# B&R Automation Studio project Cognex_V1_5
Automation Studio 4.0.21.35 SP

## Configuration PP500_15

CPU , AutomationRuntime H4.06, Build 4.1.2, Vc V4.05.6, Safety 1.6

### Hardware
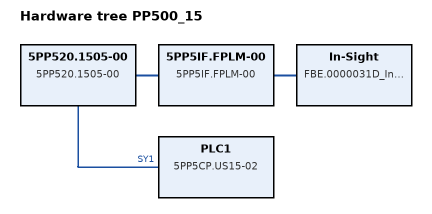
```
5PP520.1505-00 : 5PP520.1505-00 v2.0.1.1
  Connector IF3:
    ActivateDevice = 1
    Mode = DHCP Server
    InternetAddress = 192.168.0.10
    SubnetMask = 255.255.255.0
    Lease1
    LeaseName1 = loc
    LeaseStartAddress1 = 192.168.0.220
    LeaseStopAddress1 = 192.168.0.230
    LeaseSubnetMask1 = 255.255.255.0
    Vnc1
    VncVcObjectName1 = Visu
    VncPortNumber1 = 5900
    VncMaxConnections1 = 1
    VncRefreshRate1 = 1000
    VncConnectionTimeout1 = 4
    VncAuthentication1 = 1
    VncPasswordViewOnly1 = r
    VncPasswordViewControl1 = w
  VcObjectName = Visu
5PP5IF.FPLM-00 : 5PP5IF.FPLM-00 v2.1.3.0  [SL -> 5PP520.1505-00.SL1]
  Connector IF1:
    MtuSize = 1500
    CycleTime = 400
    InternetAddress = 10.49.40.10
    SubnetMask = 255.255.255.0
In-Sight : FBE.0000031D_In-Sight-7000 v1.0 (OrderNumber=In-Sight)  [PLK1 -> 5PP5IF.FPLM-00.IF1 (NodeNumber=1)]
  Supervision = off
  p2000s01_direction = wo
  p2000s02_direction = wo
  p2001s01_direction = ro
  p2001s02_direction = ro
  p2010s01_direction = ro
  p2011s01_direction = ro
  p2011s02_direction = ro
  p2011s03_direction = ro
  p2011s04_direction = ro
  p2011s05_direction = ro
  p2011s06_direction = ro
  p2011s07_direction = ro
  p2011s08_direction = ro
  p2011s09_direction = ro
  p2011s0A_direction = ro
  p2011s0B_direction = ro
  p2021s01_direction = wo
  p2021s02_direction = wo
  p2021s03_direction = wo
PLC1 : 5PP5CP.US15-02 v2.0.3.0  [SY -> 5PP520.1505-00.SY1]
  PreserveNonVolatileSystemSettings = 0
  Connections = 8
  TimerDeviceType = EPLX2X
  TaskClassIdleTime = 800
  Cyclic1Duration = 2000
  Cyclic1Tolerance = 2000
  Cyclic1Stack = 65535
  Cyclic2Stack = 65535
  Cyclic3Stack = 65535
  Cyclic4Stack = 65535
  Cyclic5Stack = 65535
  Cyclic6Stack = 65535
  Cyclic7Stack = 65535
  Cyclic8Duration = 4000
  Cyclic8Stack = 65535
  TimerDevice = 5PP5IF.FPLM-00.IF1
```

## Configuration X20CPU1484

CPU , AutomationRuntime V3.08, Build 4.1.2, Vc V3.95.6

## Logical view

Binary libraries used (declarations not repeated): Operator, Runtime, AsTime, AsIecCon, sys_lib, asstring, FileIO, Visapi, AsTCP, AsICMP, standard, BR_ATL_LOG, BR_ATL_BMP, BR_ATL_COG


- Program Logical/Cognex (IEC) - Cognex IO mapping (no source held here)

### Program Logical/CognexVisCommissioning (IEC) - Cognex camera commissioning

#### CognexVisCommissioning.var
```iecst
(*-------------------------------------------------------------------------------------------------------------------------------------------------------------------------------------------------------------------------*)
VAR
	data : ARRAY[0..999] OF USINT; (*Send and receive buffer (size must be even)*)
	data_string : ARRAY[0..19] OF STRING[80]; (*Receive data split up as string*)
	NativeModeCommandStatus : INT;
	NaticeModeCommand : USINT;
	NativeModeCommand_0 : NativeModeCommand;
	NativeModeWriteFile_0 : NativeModeWriteFile;
	DirCreate_0 : DirCreate;
	DevLink_0 : DevLink;
	TransferProgressStatus : UINT;
	vsTransferProgress : USINT;
END_VAR
(*--------------------------------------------------------------------------------------------------------------------------------------------------------------------------------------------------------------------------------------------*)
VAR
	vkNativeModeConnect : BOOL;
	NativeModeLoggedIn : UINT;
	NativeModeStatus : UINT;
	NativeModeLogin_0 : NativeModeLogin;
	NativeModeLogout_0 : NativeModeLogout;
END_VAR
(*--------------------------------------------------------------------------------------------------------------------------------------------------------------------------------------------------------------------------------------------*)
VAR
	vkTransferWrite : USINT;
	vsErrorReset : UINT := 1;
	vkErrorReset : BOOL;
END_VAR
```

#### CognexVisCommissioning.ab
```automation-basic
(********************************************************************
 * COPYRIGHT --
 ********************************************************************
 * Author: strickers
 * Version: 1.0
 * This task has the following purpose
 * - Connect to Cognex telnet (Native interface)
 * - Read command_status information
 * - Read and write camera jobs
 * - Read and write camera settings
 ********************************************************************)

PROGRAM _INIT
	(* --------------------------------------------------------------------------------------------------------- *)
	(* Create file device for Cognex files and configuration files *)
	LOOP
		DevLink_0.enable 	= 1
		DevLink_0.pDevice 	= ADR("root")
		DevLink_0.pParam 	= ADR("/DEVICE=C:\\")
		DevLink_0 FUB DevLink()
		EXITIF(DevLink_0.status <> 65535)
	ENDLOOP
	(* --------------------------------------------------------------------------------------------------------- *)
	(* Create folder for Cognex files and configuration files *)
	LOOP
		DirCreate_0.enable 	= 1
		DirCreate_0.pDevice = ADR("root")
		DirCreate_0.pName 	= ADR("cognex_files")
		DirCreate_0 FUB DirCreate()
		EXITIF(DirCreate_0.status <> 65535)
	ENDLOOP
	(* --------------------------------------------------------------------------------------------------------- *)
	(* Create file device for Cognex files and configuration files *)
	LOOP
		DevLink_0.enable 	= 1
		DevLink_0.pDevice 	= ADR("CognexFiles")
		DevLink_0.pParam 	= ADR("/DEVICE=C:\\cognex_files")
		DevLink_0 FUB DevLink()
		EXITIF(DevLink_0.status <> 65535)
	ENDLOOP
	NativeModeStatus = VIS_INACTIVE
	TransferProgressStatus = VIS_HIDDEN
END_PROGRAM

PROGRAM _CYCLIC

(* --------------------------------------------------------------------------------------------------------- *)
(* Connect to camera
(* --------------------------------------------------------------------------------------------------------- *)
IF(EDGEPOS(vkNativeModeConnect)) THEN
	NewLogEntry("Connecting to camera...", ADR(logbook), 20)
ENDIF
IF(vkNativeModeConnect = TRUE) THEN
	IF(NativeModeLoggedIn = FALSE) THEN
		NativeModeLogin_0.enable = 1
		NativeModeLogin_0.ip = ADR(CognexEthIP)
		NativeModeLogin_0 FUB NativeModeLogin()
		IF(NativeModeLogin_0.status <> 65535) THEN
			IF(NativeModeLogin_0.status = 0) THEN
				NewLogEntry("Loggged into camera", ADR(logbook), 20)
				NativeModeLoggedIn	= TRUE
				NativeModeStatus 	= VIS_ACTIVE
				NaticeModeCommand 	= CMD_SET_OFFLINE
			ELSE
				NewLogEntry("Failed to log into camera", ADR(logbook), 20)
				NativeModeStatus 	= VIS_INACTIVE
				vsErrorReset 		= VIS_ACTIVE
			ENDIF
			vkNativeModeConnect = FALSE
		endif
	ELSE
(* --------------------------------------------------------------------------------------------------------- *)
(* Disconnect from camera
(* --------------------------------------------------------------------------------------------------------- *)
		NativeModeLogout_0.enable = 1
		NativeModeLogout_0.ident = NativeModeLogin_0.ident
		NativeModeLogout_0 FUB NativeModeLogout()
		IF(NativeModeLogout_0.status <> 65535) THEN
			NewLogEntry("Loggged out of camera", ADR(logbook), 20)
			NativeModeWriteFile_0.enable = 0
			NativeModeWriteFile_0 FUB NativeModeWriteFile()

			vsTransferProgress 		= 0
			TransferProgressStatus  = VIS_HIDDEN
			vkTransferWrite 		= NONE

			NativeModeLogin_0.enable = 0
			NativeModeLogin_0 FUB NativeModeLogin()
			NativeModeStatus 	= VIS_INACTIVE
			NativeModeLoggedIn	= FALSE
			vkNativeModeConnect	= FALSE
		ENDIF
	ENDIF
ENDIF

(* --------------------------------------------------------------------------------------------------------- *)
(* Use command interface for Cognex camera
(* --------------------------------------------------------------------------------------------------------- *)
IF EDGEPOS(NaticeModeCommand = CMD_SET_OFFLINE) THEN
	NativeModeCommand_0.command = ADR("SO0")
	NewLogEntry("Set camera offline", ADR(logbook), 20)
ENDIF
IF(NaticeModeCommand <> NONE) THEN
	NativeModeCommand_0.enable 		= 1
	NativeModeCommand_0.ident 		= NativeModeLogin_0.ident
	NativeModeCommand_0.out_data 	= ADR(data)
	NativeModeCommand_0.out_size 	= SIZEOF(data)
	NativeModeCommand_0 FUB NativeModeCommand()
	NativeModeStatus = VIS_INACTIVE
	IF(NativeModeCommand_0.status <> 65535) THEN
		IF(NativeModeCommand_0.status = 0) THEN
			NewLogEntry("Command finished", ADR(logbook), 20)
			(* Separate data stream by \r\n and split into strings *)
			NativeModeCommandStatus = NativeModeSeparateData(ADR(data), NativeModeCommand_0.in_size, ADR(data_string), SIZEOF(data_string[0]), SIZEOF(data_string)/SIZEOF(data_string[0]))
			(* Check camera responds (1 = The command was executed successfully. 0=Unrecognized command. -2=The command could not be executed. *)
 			IF(NativeModeCommandStatus = 1) THEN
				NativeModeStatus = VIS_ACTIVE
			ELSE
				NewLogEntry("Camera responded with error", ADR(logbook), 20)
				vsErrorReset = VIS_ACTIVE
			ENDIF
		ELSE
			NewLogEntry("Command failed", ADR(logbook), 20)
			vsErrorReset = VIS_ACTIVE
		ENDIF
		NaticeModeCommand = NONE
	ENDIF
ENDIF

(* --------------------------------------------------------------------------------------------------------- *)
(* Write file to Cognex camera
(* --------------------------------------------------------------------------------------------------------- *)
IF EDGEPOS(vkTransferWrite = WRITE_ID1) THEN
	NativeModeWriteFile_0.command 	= ADR("WJ1")
	NativeModeWriteFile_0.file_name = ADR("1_Powerlink.job")
	NewLogEntry("Write job file ID1", ADR(logbook), 20)
ENDIF
IF EDGEPOS(vkTransferWrite = WRITE_ID2) THEN
	NativeModeWriteFile_0.command 	= ADR("WJ2")
	NativeModeWriteFile_0.file_name = ADR("2_Powerlink.job")
	NewLogEntry("Write job file ID2", ADR(logbook), 20)
ENDIF
IF EDGEPOS(vkTransferWrite = WRITE_CFG) THEN
	NativeModeWriteFile_0.command 	= ADR("WS")
	NativeModeWriteFile_0.file_name = ADR("proc.set")
	NewLogEntry("Write configuration file", ADR(logbook), 20)
ENDIF
IF(vkTransferWrite <> NONE) THEN
	NativeModeWriteFile_0.enable 	= 1
	NativeModeWriteFile_0.ident 	= NativeModeLogin_0.ident
	NativeModeWriteFile_0.device 	= ADR("CognexFiles")
	NativeModeWriteFile_0 FUB NativeModeWriteFile()
	vsTransferProgress 		= NativeModeWriteFile_0.progress
	TransferProgressStatus  = VIS_ACTIVE
	NativeModeStatus 		= VIS_INACTIVE
	IF(NativeModeWriteFile_0.status <> 65535) THEN
		IF(NativeModeWriteFile_0.status = 0) THEN
			NewLogEntry("Write file finished", ADR(logbook), 20)
			NativeModeStatus = VIS_ACTIVE
		ELSE
			NewLogEntry("Write file failed", ADR(logbook), 20)
			vsErrorReset = VIS_ACTIVE
		ENDIF
		TransferProgressStatus = VIS_HIDDEN
		vkTransferWrite = NONE
	ENDIF
ENDIF

(* --------------------------------------------------------------------------------------------------------- *)
(* Error handling and reset
(* --------------------------------------------------------------------------------------------------------- *)
IF (vkErrorReset) THEN
	IF(NativeModeLogin_0.status <> 0) THEN
		NativeModeLogin_0.enable = 0
		NativeModeLogin_0 FUB NativeModeLogin()
		NativeModeLogout_0.enable = 1
		NativeModeLogout_0.ident = NativeModeLogin_0.ident
		NativeModeLogout_0 FUB NativeModeLogout()
	ENDIF
	vsTransferProgress = 0
	vkNativeModeConnect = FALSE
	NativeModeWriteFile_0.enable = 0
	NativeModeWriteFile_0 FUB NativeModeWriteFile()
	NativeModeCommand_0.enable = 0
	NativeModeCommand_0 FUB NativeModeCommand()
	memset(ADR(logbook), 0, SIZEOF(logbook))
	NativeModeStatus 	= VIS_INACTIVE
	vsErrorReset 		= VIS_HIDDEN
	vkErrorReset 		= 0
ENDIF

END_PROGRAM
```

### Program Logical/CognexVisNativeMode (IEC) - Cognex telnet communication

#### CognexVisNativeMode.var
```iecst
(*-------------------------------------------------------------------------------------------------------------------------------------------------------------------------------------------------------------------------*)
VAR
	data : ARRAY[0..999] OF USINT; (*Send and receive buffer (size must be even)*)
	data_string : ARRAY[0..19] OF STRING[80]; (*Receive data split up as string*)
	NativeModeCommandStatus : INT;
	NaticeModeCommand : USINT;
	NativeModeCommand_0 : NativeModeCommand;
	NativeModeReadFile_0 : NativeModeReadFile;
	NativeModeWriteFile_0 : NativeModeWriteFile;
	DirCreate_0 : DirCreate;
	DevLink_0 : DevLink;
	vsTransferProgress : USINT;
	TransferProgressStatus : UINT;
END_VAR
(*--------------------------------------------------------------------------------------------------------------------------------------------------------------------------------------------------------------------------------------------*)
VAR
	vkNativeModeConnect : BOOL;
	CognexPlkIP : STRING[30] := '192.168.101.'; (*IP address for camera when connected to Ethernet port*)
	NativeModeLoggedIn : UINT;
	NativeModeStatus : UINT;
	NativeModeLogin_0 : NativeModeLogin;
	NativeModeLogout_0 : NativeModeLogout;
END_VAR
(*--------------------------------------------------------------------------------------------------------------------------------------------------------------------------------------------------------------------------------------------*)
VAR
	vkTransferCancel : BOOL;
	vkTransferRead : USINT;
	vkTransferWrite : USINT;
	vsErrorReset : UINT := 1;
	vkErrorReset : BOOL;
END_VAR
```

- Program Logical/CognexVisArchive (IEC) - Cognex picture archive (no source held here)

### Program Logical/CognexVisMain (IEC) - Cognex main visualization

#### CognexVisMain.ab
```automation-basic
(********************************************************************
 * COPYRIGHT --
 ********************************************************************
 * Author: strickers
 * Version: 1.0
 * This task has the following purpose
 * - Maintain a logbook with events coming from the camera
 * - Check the directory \Cognex for new pictures from the camera
 * - Convert the pictures from 8 Bit to 24 Bit so that they can be
 *   displayed in Visual Components
 * - Limit the amount of pictures and delete old if necessary
 * - Show picture archive and display old pictures
 * - Handle basic VC tasks like show/hide objects etc.
 ********************************************************************)

PROGRAM _INIT
	(* --------------------------------------------------------------------------------------------------------- *)
	(* Create file device for Cognex files and configuration files *)
	LOOP
		DevLink_0.enable 	= 1
		DevLink_0.pDevice 	= ADR("root")
		DevLink_0.pParam 	= ADR("/DEVICE=C:\\")
		DevLink_0 FUB DevLink()
		EXITIF(DevLink_0.status <> 65535)
	ENDLOOP
	(* --------------------------------------------------------------------------------------------------------- *)
	(* Create cognex folder for bitmaps on boot up *)
	LOOP
		DirCreate_0.enable 	= 1
		DirCreate_0.pDevice = ADR("root")
		DirCreate_0.pName 	= ADR("cognex_pics")
		DirCreate_0 FUB DirCreate()
		EXITIF(DirCreate_0.status <> 65535)
	ENDLOOP
	(* --------------------------------------------------------------------------------------------------------- *)
	(* Create file device for Cognex files and configuration files *)
	LOOP
		DevLink_0.enable 	= 1
		DevLink_0.pDevice 	= ADR("CognexPictures")
		DevLink_0.pParam 	= ADR("/DEVICE=C:\\cognex_pics")
		DevLink_0 FUB DevLink()
		EXITIF(DevLink_0.status <> 65535)
	ENDLOOP
	(* --------------------------------------------------------------------------------------------------------- *)
	(* Enable camera trigger, get VC handle, calculate max number of pitcures *)
	cognex_1.cmd.trigger_enable = TRUE
	cognex_1.cmd.job_id = 1
	VChandle = VA_Setup(1, "Visu")
	dir_entry_max =  SIZEOF(dir_data)/SIZEOF(dir_data[0])-1
END_PROGRAM

PROGRAM _CYCLIC
	(* --------------------------------------------------------------------------------------------------------- *)
	(* Enable/Disable vis object depending on cemera status connected, online ... *)
	(* --------------------------------------------------------------------------------------------------------- *)
	vsCameraConnectedPlk = UINT(NOT cognex_1.sta.connected_plk)*2
	vsCameraOnline = UINT(NOT cognex_1.sta.connected_plk OR NOT cognex_1.sta.online)*2
	vsCameraTrigger = UINT(NOT cognex_1.sta.connected_plk OR NOT cognex_1.sta.online OR NOT cognex_1.sta.trigger_ready OR (step_pic <> 0))*2
	vsCameraChangeJob = UINT(NOT cognex_1.sta.connected_plk OR cognex_1.sta.online)*2
	IF(edgeneg(cognex_1.sta.job_loading)) THEN
		IF(cognex_1.sta.job_id = 1) THEN
			vsCameraJob1 = VIS_ACTIVE
		ELSE
			vsCameraJob1 = VIS_HIDDEN
		ENDIF
	ENDIF

	(* --------------------------------------------------------------------------------------------------------- *)
	(* Display camera pictures and maintain max number of pictures *)
	(* --------------------------------------------------------------------------------------------------------- *)
	CASE step_pic OF
		(* --------------------------------------------------------------------------------------------------------- *)
		ACTION STP_INIT:
			(* When new camera trigger is fired, create time stamp to detect new pictures, add 2 second tolerance *)
			IF cognex_1.cmd.trigger THEN
				cognex_1.cmd.trigger = 0
				DTGetTime_0.enable = 1
				DTGetTime_0 FUB DTGetTime()
				DTGetTimeTollerance = UDINT(DTGetTime_0.DT1)
				DTGetTimeTollerance = DTGetTimeTollerance - 2
				DTnow = DT(DTGetTimeTollerance)
				step_pic = STP_RESULT
			ENDIF
		ENDACTION
		(* --------------------------------------------------------------------------------------------------------- *)
		ACTION STP_RESULT:
			(* When new result arrives, ceate lofg entry, load default values, erase previous picture *)
			IF EDGEPOS(cognex_1.sta.results_valid) THEN
				NewLogEntry("Looking for new picture", ADR(logbook), 20)
				dir_wait_time 	= 0
				dir_entry 		= 0
				TON_10ms_0.IN 	= 0
				TON_10ms_0 FUB TON_10ms()
				step_pic = STP_WAIT
			ENDIF
		ENDACTION
		(* --------------------------------------------------------------------------------------------------------- *)
		ACTION STP_WAIT:
			(* Erase old picture *)
			IF(VA_Saccess(1, VChandle) = 0) THEN
				VCerror = VA_Rect(1, VChandle, 70, 505, PictureWidth, PictureHeight, 7, 0)
				VA_Srelease(1, VChandle)
			ENDIF
			(* The camera needs time to store the picture on the PLC. Check after 0.5s if new picture arrived *)
			TON_10ms_0.IN = 1
			TON_10ms_0.PT = 50
			TON_10ms_0 FUB TON_10ms()
			IF(TON_10ms_0.Q) THEN
				step_pic = STP_DIR_READ
			ENDIF
		ENDACTION
		(* --------------------------------------------------------------------------------------------------------- *)
		ACTION STP_DIR_READ:
			(* Read all file names and date stamps from directory *)
			DirRead_0.enable 	= 1
			DirRead_0.pDevice 	= ADR("CognexPictures")
			DirRead_0.entry 	= dir_entry
			DirRead_0.option 	= fiFILE
			DirRead_0.pData 	= ADR(dir_data[dir_entry])
			DirRead_0.data_len 	= SIZEOF(dir_data[dir_entry])
			DirRead_0 FUB DirRead()

			(* Stop reading files when max number is reached *)
			IF (DirRead_0.status = fiERR_NO_MORE_ENTRIES) OR ((DirRead_0.status = 0) AND (dir_entry = dir_entry_max)) THEN
				step_pic = STP_DIR_EVAL
			(* Its all good, read next entry *)
			ELSE IF DirRead_0.status = 0 THEN
				dir_entry = dir_entry + 1
			(* Jump to error step when FB faults *)
			ELSE IF (DirRead_0.status <> 65535) THEN
				NewLogEntry("#Error: dir read", ADR(logbook), 20)
				step_pic = STP_ERROR
			ENDIF
		ENDACTION
		(* --------------------------------------------------------------------------------------------------------- *)
		ACTION STP_DIR_EVAL:
			(* Make sure we have at least one file entry, jump to wait state and wait another 0.5s before checking again *)
			IF (dir_entry = 0) THEN
				IF (dir_wait_time < dir_timeout) THEN
					dir_wait_time = dir_wait_time + TON_10ms_0.PT*10
					dir_entry = 0
					TON_10ms_0.IN = 0
					TON_10ms_0 FUB TON_10ms()
					step_pic = STP_WAIT
				(* Give up after timeout when no picture was found *)
				ELSE
					NewLogEntry("No new picture found", ADR(logbook), 20)
					step_pic = STP_INIT
				ENDIF
			ELSE
				(* Search for newest file to display and oldest file to delete *)
				memcpy(ADR(dir_data_newest), ADR(dir_data[0]), SIZEOF(dir_data_newest))
				memcpy(ADR(dir_data_oldest), ADR(dir_data[0]), SIZEOF(dir_data_oldest))
				LOOP x=1 TO dir_entry-1 DO
					IF((dir_data_newest.Date < dir_data[x].Date) AND (memcmp(ADR(dir_data[x].Filename), ADR("brplc"), 5) = 0)) THEN
						memcpy(ADR(dir_data_newest), ADR(dir_data[x]), SIZEOF(dir_data_newest))
					ENDIF
					IF(dir_data_oldest.Date > dir_data[x].Date) THEN
						memcpy(ADR(dir_data_oldest), ADR(dir_data[x]), SIZEOF(dir_data_newest))
					ENDIF
				ENDLOOP
				(* When doing folder cleanup jump back to file delete *)
				IF (dir_cleanup) THEN
					step_pic = STP_BMP_CLEANUP
				(* Make sure newest file was created after trigger event *)
				ELSE IF (dir_data_newest.Date >= DTnow) THEN
					strcpy(ADR(file_newest), ADR(dir_data_newest.Filename))
					NewLogEntry("Converting bitmap...", ADR(logbook), 20)
					step_pic = STP_VC_CONVERT
				(* Jump to wait state and wait another 0.5s before checking again *)
				ELSE IF (dir_data_newest.Date < DTnow) AND (dir_wait_time < dir_timeout) THEN
					dir_wait_time = dir_wait_time + 500
					dir_entry = 0
					TON_10ms_0.IN = 0
					TON_10ms_0 FUB TON_10ms()
					step_pic = STP_WAIT
				(* Give up after timeout when no picture was found *)
				ELSE IF (dir_data_newest.Date < DTnow) AND (dir_wait_time >= dir_timeout) THEN
					NewLogEntry("No new picture found", ADR(logbook), 20)
					step_pic = STP_BMP_CLEANUP
				ENDIF
			ENDIF
		ENDACTION
		(* --------------------------------------------------------------------------------------------------------- *)
		ACTION STP_VC_CONVERT:
			(* Convert picture from 8 Bit to 24 Bit *)
			strcpy(ADR(file_converted), ADR("c"))
			strcat(ADR(file_converted), ADR(file_newest))
			BmpConvert_0.enable 			= 1
			BmpConvert_0.pDevice 			= ADR("CognexPictures")
			BmpConvert_0.pFileSource 		= ADR(file_newest)
			BmpConvert_0.pFileDestination 	= ADR(file_converted)
			BmpConvert_0 FUB BmpConvert()

			IF (BmpConvert_0.status = 0) THEN
				NewLogEntry("Converting done", ADR(logbook), 20)
				VCbitmap_tmp = 0
				step_pic = STP_VC_LOAD
			(* Jump to error step when FB faults *)
			ELSE IF (BmpConvert_0.status <> 65535) THEN
				NewLogEntry("#Error: convert bitmap", ADR(logbook), 20)
				step_pic = STP_ERROR
			ENDIF
		ENDACTION
		(* --------------------------------------------------------------------------------------------------------- *)
		ACTION STP_VC_LOAD:
			(* Load picture into memory *)
			IF(VA_Saccess(1, VChandle) = 0) THEN
				VCerror = VA_LoadBitmap(1, VChandle, "CognexPictures", file_converted, ADR(VCbitmap_tmp))
				IF(VCerror = 0) THEN
					VCbitmap ACCESS VCbitmap_tmp
					step_pic = STP_VC_SHOW
				ELSE IF (VCerror <> 7000) THEN
					NewLogEntry("#Error: load bitmap", ADR(logbook), 20)
					step_pic = STP_ERROR
				ENDIF
				VA_Srelease(1, VChandle)
			ENDIF
		ENDACTION
		(* --------------------------------------------------------------------------------------------------------- *)
		ACTION STP_VC_SHOW:
			(* Display new picture *)
			IF(VA_Saccess(1, VChandle) = 0) THEN
				VCerror = VA_BlitBitmap(1, VChandle, ADR(VCbitmap), 70, 505, 70, 505, 70+PictureWidth, 505+PictureHeight, 1)
				IF(VCerror = 0) THEN
					VCbitmap ACCESS VCbitmap_tmp
					step_pic = STP_VC_FREE
				ELSE IF (VCerror <> 7000) THEN
					NewLogEntry("#Error: show bitmap", ADR(logbook), 20)
					step_pic = STP_ERROR
				ENDIF
				VA_Srelease(1, VChandle)
			ENDIF
		ENDACTION
		(* --------------------------------------------------------------------------------------------------------- *)
		ACTION STP_VC_FREE:
			(* Free up memory *)
			IF(VA_Saccess(1, VChandle) = 0) THEN
				VCerror = VA_FreeBitmap(1, VChandle, ADR(VCbitmap_tmp))
				IF(VCerror = 0) THEN
					VCbitmap ACCESS VCbitmap_tmp
					step_pic = STP_BMP_DELETE
				ELSE IF (VCerror <> 7000) then
					NewLogEntry("#Error: free bitmap", ADR(logbook), 20)
					step_pic = STP_ERROR
				ENDIF
				VA_Srelease(1, VChandle)
			ENDIF
		ENDACTION
		(* --------------------------------------------------------------------------------------------------------- *)
		ACTION STP_BMP_DELETE:
			(* Delete old converted picture *)
			FileDelete_0.enable 	= 1
			FileDelete_0.pDevice 	= ADR("CognexPictures")
			FileDelete_0.pName 		= ADR(file_newest)
			FileDelete_0 FUB FileDelete()

			IF (FileDelete_0.status <> 65535) THEN
				step_pic = STP_BMP_CLEANUP
			ENDIF
		ENDACTION
		(* --------------------------------------------------------------------------------------------------------- *)
		ACTION STP_BMP_CLEANUP:
			(* Make sure we limit the number of pictures and delete oldest if necessary *)
			IF (dir_entry < dir_entry_max) THEN
				dir_cleanup = FALSE
				step_pic = STP_INIT
			ELSE
				FileDelete_0.enable 	= 1
				FileDelete_0.pDevice 	= ADR("CognexPictures")
				FileDelete_0.pName 		= ADR(dir_data_oldest.Filename)
				FileDelete_0 FUB FileDelete()
				IF (FileDelete_0.status <> 65535) THEN
					dir_entry	= 0
					dir_cleanup = TRUE
					step_pic = STP_DIR_READ
				ENDIF
			ENDIF
		ENDACTION
		(* --------------------------------------------------------------------------------------------------------- *)
		ACTION STP_ERROR:
			vsErrorReset = 0
			BmpConvert_0.enable = 0
			BmpConvert_0 FUB BmpConvert()
			IF (vkErrorReset) THEN
				memset(ADR(logbook), 0, SIZEOF(logbook))
				vsErrorReset = 1
				vkErrorReset = 0
				step_pic = STP_INIT
			ENDIF
		ENDACTION
	ENDCASE
END_PROGRAM
```

- Visualisation Logical/Visu (not shown)

Listed in the project but not available here: Logical/Global.typ, Logical/Global.var, Logical/AdditionalFiles, Logical/Cognex/Cognex.ab, Logical/Cognex/Cognex.typ, Logical/Cognex/Cognex.var, Logical/CognexVisArchive/CognexVisArchive.ab, Logical/CognexVisArchive/CognexVisArchive.typ, Logical/CognexVisArchive/CognexVisArchive.var
